SUBAPPLICATION LED_Test (* Subapplication Type *)
  (* Standard: 61499-2 *)
  (* Version 1.0, 2023-10-23, franz *)
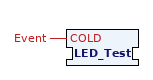
  EVENT_INPUT
    COLD;
  END_EVENT
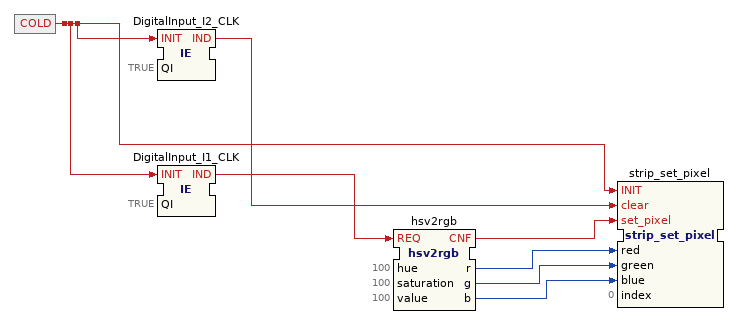
  FBS
    DigitalInput_I1_CLK : IE(QI := TRUE);
    DigitalInput_I2_CLK : IE(QI := TRUE);
    strip_set_pixel : strip_set_pixel(index := 0);
    hsv2rgb : hsv2rgb(hue := 100, saturation := 100, value := 100);
  END_FBS
  EVENT_CONNECTIONS
    COLD TO DigitalInput_I1_CLK.INIT;
    COLD TO DigitalInput_I2_CLK.INIT;
    COLD TO strip_set_pixel.INIT;
    DigitalInput_I2_CLK.IND TO strip_set_pixel.clear;
    hsv2rgb.CNF TO strip_set_pixel.set_pixel;
    DigitalInput_I1_CLK.IND TO hsv2rgb.REQ;
  END_CONNECTIONS
  DATA_CONNECTIONS
    hsv2rgb.r TO strip_set_pixel.red;
    hsv2rgb.g TO strip_set_pixel.green;
    hsv2rgb.b TO strip_set_pixel.blue;
  END_CONNECTIONS
END_SUBAPPLICATION
